FUNCTION_BLOCK StateSuspended EXTENDS _AbstractState
VAR_INPUT
END_VAR
VAR_OUTPUT
END_VAR
VAR
	_bSuspendLock: BOOL;
END_VAR

(*
Determines whether the state can be activated.  
Returns `TRUE` by default but can be overridden for specific activation conditions.
*)
METHOD PROTECTED CanActivate : BOOL
CanActivate := _ctx.smgr.Current.Tag = _ctx.execute.Tag;
END_METHOD

(*
Executed when the state is entered.  
Provides a hook for defining state-specific behavior to be performed during the transition into this state.
*)
METHOD PROTECTED OnEntry
_ctx.sHmiStatusText := 'Suspended: I guess we wait... ';
END_METHOD

END_FUNCTION_BLOCK

(* stored: Version 1.1.0.1
   POU StateSuspended: Id {e30e6341-c6bb-48e9-97d2-f8746561be2b}, SpecialFunc None
   Method CanActivate: Id {070cfb98-766f-4eb7-bc81-754ff7cee900}
   Method OnEntry: Id {db54bebc-aa27-4ae2-93ae-230efa966949} *)
